TYPE ST_SCANNER_CameraMap :
STRUCT
	nIndex				: INT;
	nReqProgram			: BYTE;
	stOptions				: ST_SCANNER_Options;
	aPackPos				: ARRAY[1..5, 1..cMAX_CAMERA_PROG_NUMBER] OF BYTE;
	aTargetBuffer			: ARRAY[1..5] OF BYTE;

END_STRUCT
END_TYPE

(* stored: Version 1.1.0.1, ProductVersion 3.1.4024.15
   DUT ST_SCANNER_CameraMap: Id {01a09907-4501-4a29-8248-d6afb1c08981} *)
